DATA_BLOCK "Pilz_fb_DB"
{ S7_Optimized_Access := 'FALSE' }
VERSION : 0.1
NON_RETAIN
// ATTRIBUTES
// AUTO_NUMBER = False
// BLOCK_NUMBER = 2700
// END_ATTRIBUTES
"Pilz_fb"

BEGIN

END_DATA_BLOCK

